FUNCTION_BLOCK A2X_AUI_DEMUX_5 (* A2X demultiplexor (generic FB) Adapter-Ausgang wird nur bei Wertänderung aktualisiert (Event nur bei tatsächlicher Änderung). *)
  (* Standard: 61499-2; Description: Copyright (c) 2026 Meisterschulen am Ostbahnhof This program and the accompanying materials are made available under the terms of the Eclipse Public License 2.0 which is available at https://www.eclipse.org/legal/epl-2.0/ SPDX-License-Identifier: EPL-2.0 *)
  (* Version 1.0, 2026-09-11, Franz Höpfinger, Meisterschulen am Ostbahnhof, A2X-Variante von AX_AUI_DEMUX_5 - Adapter-Backend GEN_A2X_AUI_DEMUX noch zu implementieren. *)
  PACKAGE adapter::selection::unidirectional;
  {SET_ATTRIBUTE(eclipse4diac::core::GenericClassName, 'GEN_A2X_AUI_DEMUX')}
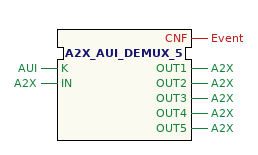
  EVENT_OUTPUT
    CNF; (* Confirmation of Set Index K *)
  END_EVENT
  SOCKETS
    K : adapter::types::unidirectional::AUI; (* index *)
    IN : adapter::types::unidirectional::A2X; (* Input Value to demultiplex *)
  END_SOCKETS
  PLUGS
    OUT1 : adapter::types::unidirectional::A2X; (* Output value 1 (selected when K = 0) *)
    OUT2 : adapter::types::unidirectional::A2X; (* Output value 2 (selected when K = 1) *)
    OUT3 : adapter::types::unidirectional::A2X; (* Output value 3 (selected when K = 2) *)
    OUT4 : adapter::types::unidirectional::A2X; (* Output value 4 (selected when K = 3) *)
    OUT5 : adapter::types::unidirectional::A2X; (* Output value 5 (selected when K = 4) *)
  END_PLUGS
END_FUNCTION_BLOCK
